// TIA Portal V16 export
// export: Created 2021-12-08T06:27:39.9823919Z, ExportSetting WithDefaults, DisplayName Totally Integrated Automation Portal, DisplayVersion V16 Update 4, DisplayName TIA Portal Version Control Interface, DisplayVersion V16 Update 2, DisplayName TIA Portal Openness, DisplayVersion V16 Update 4, DisplayName TIA Portal Teamcenter Gateway, DisplayVersion V16, DisplayName SINAMICS Startdrive Advanced, DisplayVersion V16 Update 5, DisplayName SINAMICS Startdrive G130, G150, S120, S150, SINAMICS MV, S210, DisplayVersion V16 Update 5, DisplayName SINAMICS Startdrive G110M, G120, G120C, G120D, G120P, G115D, DisplayVersion V16 Update 5, DisplayName STEP 7 Professional, DisplayVersion V16 Update 4, DisplayName STEP 7 Safety, DisplayVersion V16, DisplayName WinCC Advanced, DisplayVersion V16 Update 4
FUNCTION_BLOCK "FB_LexiumModbusTCP"   // FB301, FBD
{ S7_Optimized_Access := 'TRUE' }
VERSION : 0.1
// stored: AutoNumber false, IsIECCheckEnabled false, IsRetainMemResEnabled false, MemoryReserve 100, SetENOAutomatically false, UDAEnableTagReadback false
   VAR_INPUT
      IP_OCTET_01 : USInt;
      IP_OCTET_2 : USInt;
      IP_OCTET_3 : USInt;
      IP_OCTET_4 : USInt;
      ConnectID_1 : CONN_OUC;
      ConnectID_2 : CONN_OUC;
      ConnectID_3 : CONN_OUC;
      ConnectID_4 : CONN_OUC;
      vix_DriveEnable : Bool;
      "vir_Increment/Meter" : Real;
      vix_ExecuteCalib : Bool;
      vii_CalibPos : Int;
      vir_Offset : Real;
      vix_OffsetEnable : Bool;
      vir_RequestPosition_mm : Real;
      vix_ExecuteAutomatic : Bool;
      vii_nVSlow : Int;
      vii_nVFast : Int := 0;
      vii_nVManual : Int := 0;
      vir_nTolerancePosition : Real := 0.0;
      vix_ManualBigger : Bool;
      vix_ManualSmaller : Bool;
      vir_MaxFormat_mm : Real;
      vir_MinFormat_mm : Real;
      vix_ManualParameterDownload : Bool;
      vix_QuickStop : Bool;
      vix_FaultReset : Bool;
   END_VAR
   VAR_OUTPUT
      vix_DriveState : Byte;
      vqx_ComOk : Bool;
      vqx_ReferenceOK : Bool;
      vqx_Error : Bool;
      vqr_ActualPosition_mm : Real;
      vqx_PositionReached : Bool;
      vqx_SoftLimitMAX : Bool;
      vqx_SoftLimitMIN : Bool;
      vqx_SwitchedOn : Bool;
      vqx_DriveFault : Bool;
      vqx_QickStopActive : Bool;
   END_VAR
   VAR_IN_OUT
      ILE_ParameterDB : "ILE1B_Parameter";
      viqr_nToleranceVSlow : Real := 0.0;
      viqr_nToleranceVFast : Real := 0.0;
   END_VAR
   VAR
      Axis_Ref { S7_SetPoint := 'True'} : "ILx2T_Ref";
      ILx2_ModbusTCP_Data_Instance { S7_SetPoint := 'True'} : "ILx2_ModbusTCP_Data";
      ILx2T_Control_Instance { S7_SetPoint := 'True'} : "ILx2T_Control";
      ILx2T_Homing_Instance { S7_SetPoint := 'True'} : "ILx2T_Homing";
      ILx2T_Jog_Instance { S7_SetPoint := 'True'} : "ILx2T_Jog";
      ILx2T_ProfilePosition_Instance { S7_SetPoint := 'True'} : "ILx2T_ProfilePosition";
      ILx2T_ProfileVelocity_Instance { S7_SetPoint := 'True'} : "ILx2T_ProfileVelocity";
      ILx2T_Parameter_Read_Write_Instance { S7_SetPoint := 'True'} : "ILx2T_Parameter_Read_Write";
      ILx2T_SetAcceleration { S7_SetPoint := 'True'} : "ILx2T_Parameter_Read_Write";
      ILx2T_SetDeceleration { S7_SetPoint := 'True'} : "ILx2T_Parameter_Read_Write";
      ILx2T_ReadActualPosition { S7_SetPoint := 'True'} : "ILx2T_Parameter_Read_Write";
      ILx2T_ReadActualVelocity { S7_SetPoint := 'True'} : "ILx2T_Parameter_Read_Write";
      vsx_ComError { S7_SetPoint := 'True'} : Bool;
      vsx_HomeError : Bool;
      vsx_JogError : Bool;
      vsx_PositionError : Bool;
      vsx_VelocityError : Bool;
      vsx_ReadWriteError1 : Bool;
      vsx_ReadWriteError2 : Bool;
      vsx_ReadWriteError3 : Bool;
      vsx_ReadWriteError4 : Bool;
      vsx_ReadWriteError5 : Bool;
      vsr_HomeRefAppPos : Real;
      vqr_RequestPosplusOffset : Real;
      vsr_RequestPosPlusOffsetLimited : Real;
      vqw_StopFaulthex : DWord;
      tmpExecuteAutoSet : Bool;
      tmpRangeMin { ExternalAccessible := 'False'; ExternalVisible := 'False'; ExternalWritable := 'False'} : Real;
      tmpRangeMax { ExternalAccessible := 'False'; ExternalVisible := 'False'; ExternalWritable := 'False'} : Real;
      P_Trig_ComOK : Bool;
      vsx_SetValueOutOfRange : Bool;
      TimerOffsetCorrectino : IEC_TIMER;
      TimerDelayParamterDownload { S7_SetPoint := 'True'} : IEC_TIMER;
      fbMaticExt_Instance { S7_SetPoint := 'True'} : "fbMaticExt";
      TargetVelocity { S7_SetPoint := 'True'} : Int;
      vsi_AcutalPosInc : DInt;
      Testbit : Bool;
   END_VAR
BEGIN

REGION Network 1: Error
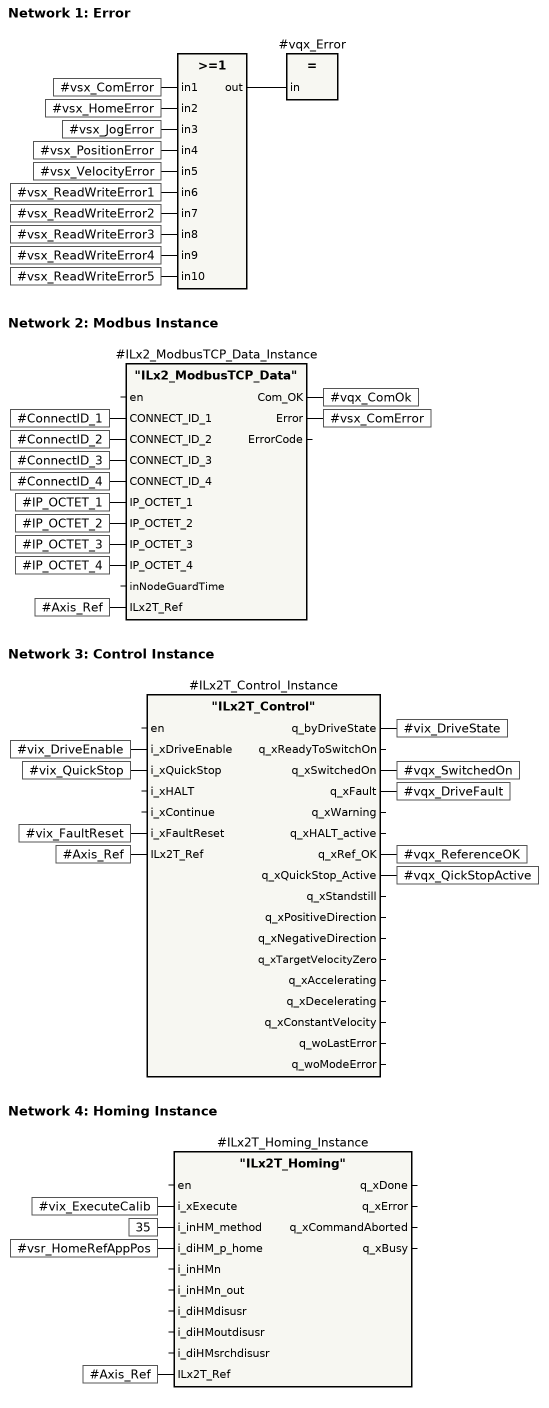
   #vqx_Error := #vsx_ComError OR #vsx_HomeError OR #vsx_JogError OR #vsx_PositionError OR #vsx_VelocityError OR #vsx_ReadWriteError1 OR #vsx_ReadWriteError2 OR #vsx_ReadWriteError3 OR #vsx_ReadWriteError4 OR #vsx_ReadWriteError5;
END_REGION

REGION Network 2: Modbus Instance
   // Error ID -TIA online help (MB_CLIENT)
   #ILx2_ModbusTCP_Data_Instance(CONNECT_ID_1 := #ConnectID_1,   // "ILx2_ModbusTCP_Data"
                           CONNECT_ID_2 := #ConnectID_2,
                           CONNECT_ID_3 := #ConnectID_3,
                           CONNECT_ID_4 := #ConnectID_4,
                           IP_OCTET_1 := #IP_OCTET_1,
                           IP_OCTET_2 := #IP_OCTET_2,
                           IP_OCTET_3 := #IP_OCTET_3,
                           IP_OCTET_4 := #IP_OCTET_4,
                           ILx2T_Ref := #Axis_Ref,
                           Com_OK => #vqx_ComOk,
                           Error => #vsx_ComError);
END_REGION

REGION Network 3: Control Instance
   #ILx2T_Control_Instance(i_xDriveEnable := #vix_DriveEnable,   // "ILx2T_Control"
                           i_xQuickStop := #vix_QuickStop,
                           i_xFaultReset := #vix_FaultReset,
                           ILx2T_Ref := #Axis_Ref,
                           q_byDriveState => #vix_DriveState,
                           q_xSwitchedOn => #vqx_SwitchedOn,
                           q_xFault => #vqx_DriveFault,
                           q_xRef_OK => #vqx_ReferenceOK,
                           q_xQuickStop_Active => #vqx_QickStopActive);
END_REGION

REGION Network 4: Homing Instance
   #ILx2T_Homing_Instance(i_xExecute := #vix_ExecuteCalib,   // "ILx2T_Homing"
                          i_inHM_method := 35,
                          i_diHM_p_home := #vsr_HomeRefAppPos,
                          ILx2T_Ref := #Axis_Ref);
END_REGION

REGION Network 5: Jog Instance (Not Used)
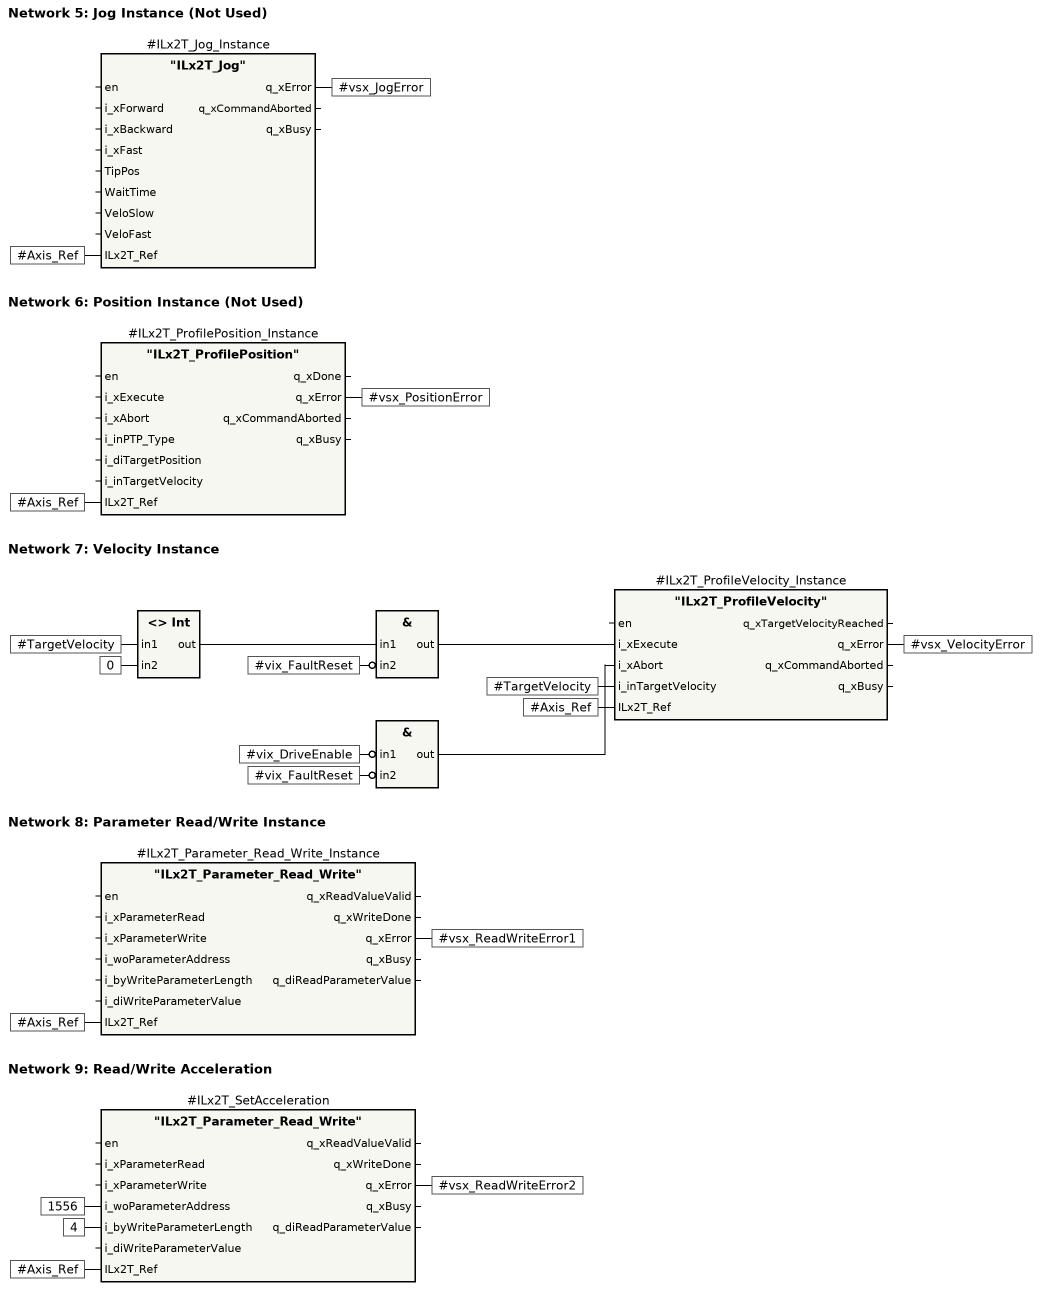
   #ILx2T_Jog_Instance(ILx2T_Ref := #Axis_Ref, q_xError => #vsx_JogError);   // "ILx2T_Jog"
END_REGION

REGION Network 6: Position Instance (Not Used)
   #ILx2T_ProfilePosition_Instance(ILx2T_Ref := #Axis_Ref, q_xError => #vsx_PositionError);   // "ILx2T_ProfilePosition"
END_REGION

REGION Network 7: Velocity Instance
   #ILx2T_ProfileVelocity_Instance(i_xExecute := (#TargetVelocity <> 0) AND NOT #vix_FaultReset,   // "ILx2T_ProfileVelocity"
                           i_xAbort := NOT #vix_DriveEnable AND NOT #vix_FaultReset,
                           i_inTargetVelocity := #TargetVelocity,
                           ILx2T_Ref := #Axis_Ref,
                           q_xError => #vsx_VelocityError);
END_REGION

REGION Network 8: Parameter Read/Write Instance
   #ILx2T_Parameter_Read_Write_Instance(ILx2T_Ref := #Axis_Ref, q_xError => #vsx_ReadWriteError1);   // "ILx2T_Parameter_Read_Write"
END_REGION

REGION Network 9: Read/Write Acceleration
   #ILx2T_SetAcceleration(i_woParameterAddress := 1556,   // "ILx2T_Parameter_Read_Write"
                          i_byWriteParameterLength := 4,
                          ILx2T_Ref := #Axis_Ref,
                          q_xError => #vsx_ReadWriteError2);
END_REGION

REGION Network 10: Read/Write Deceleration
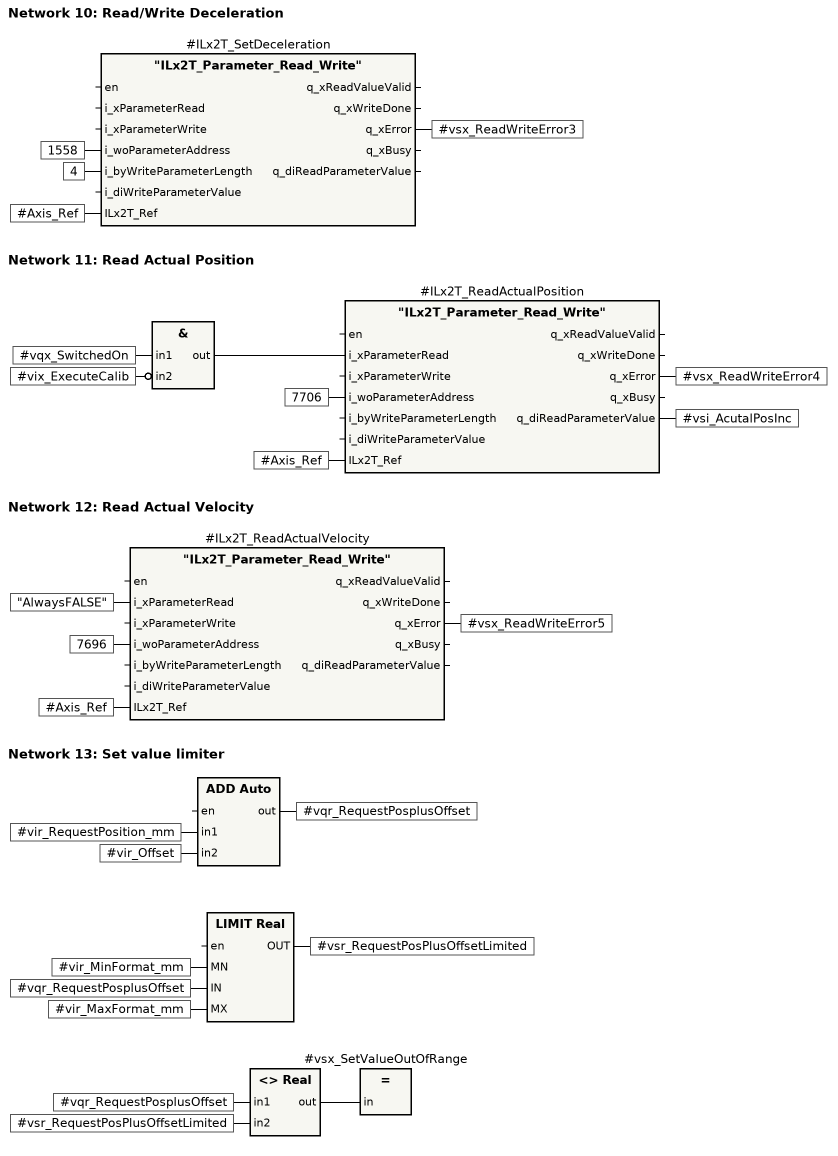
   #ILx2T_SetDeceleration(i_woParameterAddress := 1558,   // "ILx2T_Parameter_Read_Write"
                          i_byWriteParameterLength := 4,
                          ILx2T_Ref := #Axis_Ref,
                          q_xError => #vsx_ReadWriteError3);
END_REGION

REGION Network 11: Read Actual Position
   #ILx2T_ReadActualPosition(i_xParameterRead := #vqx_SwitchedOn AND NOT #vix_ExecuteCalib,   // "ILx2T_Parameter_Read_Write"
                           i_woParameterAddress := 7706,
                           ILx2T_Ref := #Axis_Ref,
                           q_xError => #vsx_ReadWriteError4,
                           q_diReadParameterValue => #vsi_AcutalPosInc);
END_REGION

REGION Network 12: Read Actual Velocity
   #ILx2T_ReadActualVelocity(i_xParameterRead := "AlwaysFALSE",   // "ILx2T_Parameter_Read_Write"
                           i_woParameterAddress := 7696,
                           ILx2T_Ref := #Axis_Ref,
                           q_xError => #vsx_ReadWriteError5);
END_REGION

REGION Network 13: Set value limiter
   #vqr_RequestPosplusOffset := #vir_RequestPosition_mm + #vir_Offset;
   #vsr_RequestPosPlusOffsetLimited := LIMIT(MN := #vir_MinFormat_mm, IN := #vqr_RequestPosplusOffset, MX := #vir_MaxFormat_mm);
   #vsx_SetValueOutOfRange := #vqr_RequestPosplusOffset <> #vsr_RequestPosPlusOffsetLimited;
END_REGION

REGION Network 14: Matic Module
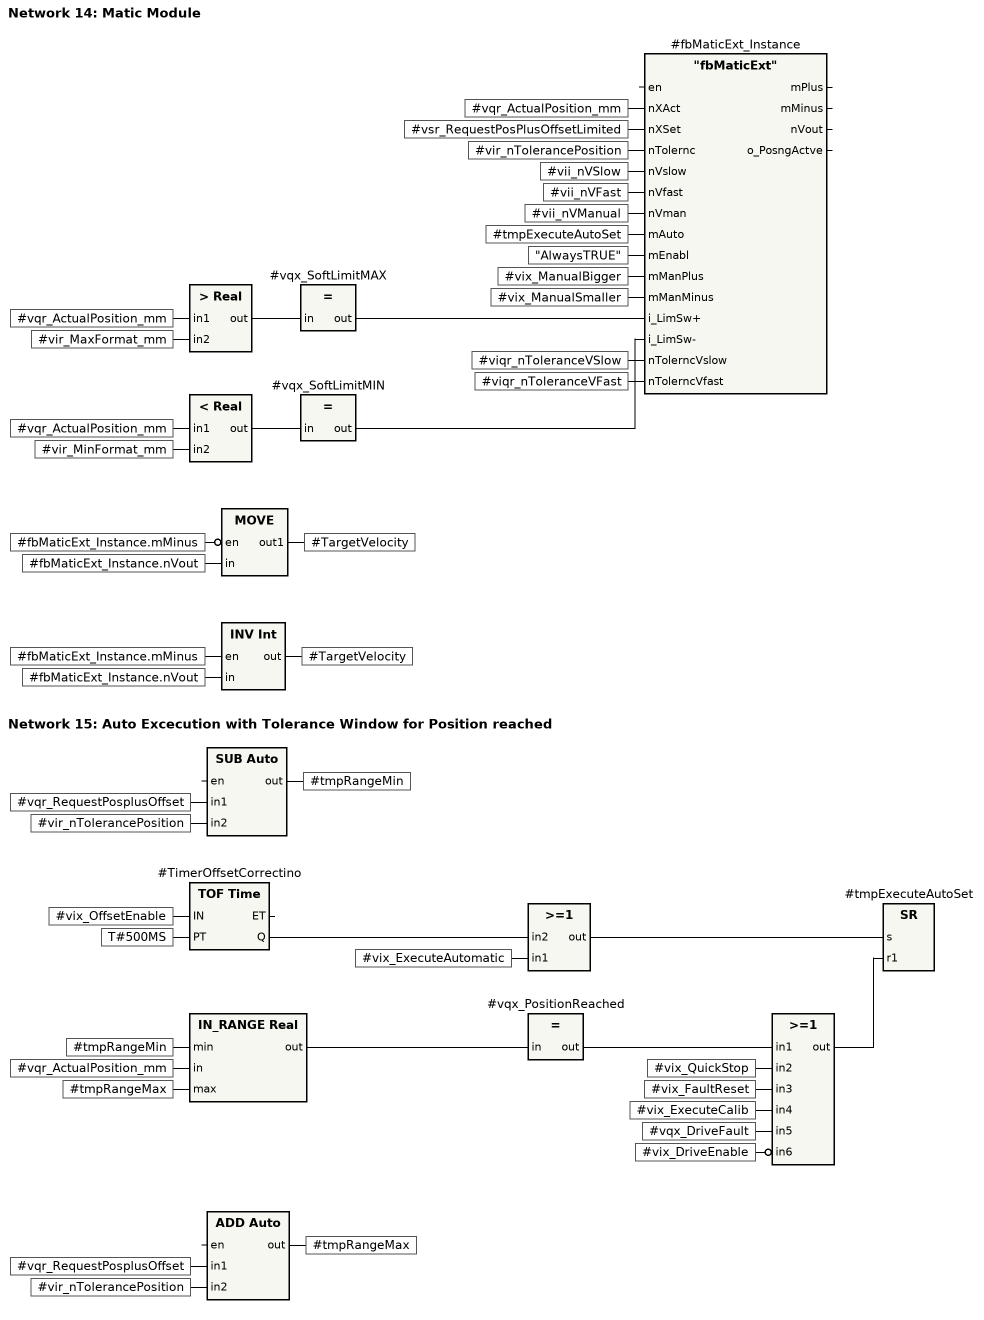
   #vqx_SoftLimitMAX := #vqr_ActualPosition_mm > #vir_MaxFormat_mm;
   #vqx_SoftLimitMIN := #vqr_ActualPosition_mm < #vir_MinFormat_mm;
   #fbMaticExt_Instance(nXAct := #vqr_ActualPosition_mm,   // "fbMaticExt"
                        nXSet := #vsr_RequestPosPlusOffsetLimited,
                        nTolernc := #vir_nTolerancePosition,
                        nVslow := #vii_nVSlow,
                        nVfast := #vii_nVFast,
                        nVman := #vii_nVManual,
                        mAuto := #tmpExecuteAutoSet,
                        mEnabl := "AlwaysTRUE",
                        mManPlus := #vix_ManualBigger,
                        mManMinus := #vix_ManualSmaller,
                        "i_LimSw+" := #vqx_SoftLimitMAX,
                        "i_LimSw-" := #vqx_SoftLimitMIN,
                        nTolerncVslow := #viqr_nToleranceVSlow,
                        nTolerncVfast := #viqr_nToleranceVFast);
   IF NOT #fbMaticExt_Instance.mMinus THEN #TargetVelocity := #fbMaticExt_Instance.nVout; END_IF;
   IF #fbMaticExt_Instance.mMinus THEN #TargetVelocity := NOT #fbMaticExt_Instance.nVout; END_IF;
END_REGION

REGION Network 15: Auto Excecution with Tolerance Window for Position reached
   #tmpRangeMin := #vqr_RequestPosplusOffset - #vir_nTolerancePosition;
   #TimerOffsetCorrectino.TOF(IN := #vix_OffsetEnable, PT := T#500MS);
   #vqx_PositionReached := (#tmpRangeMin <= #vqr_ActualPosition_mm) AND (#vqr_ActualPosition_mm <= #tmpRangeMax);
   IF #TimerOffsetCorrectino.Q OR #vix_ExecuteAutomatic THEN
       #tmpExecuteAutoSet := TRUE;   // SR flip-flop
   END_IF;
   IF #vqx_PositionReached OR #vix_QuickStop OR #vix_FaultReset OR #vix_ExecuteCalib OR #vqx_DriveFault OR NOT #vix_DriveEnable THEN
       #tmpExecuteAutoSet := FALSE;
   END_IF;
   #tmpRangeMax := #vqr_RequestPosplusOffset + #vir_nTolerancePosition;
END_REGION

REGION Network 16: Scaling Increment in mm
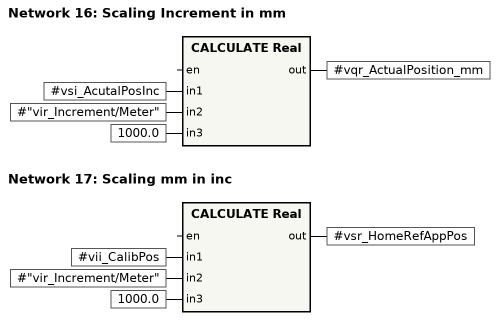
   #vqr_ActualPosition_mm := #vsi_AcutalPosInc * (#"vir_Increment/Meter"/1000.0);
END_REGION

REGION Network 17: Scaling mm in inc
   #vsr_HomeRefAppPos := #vii_CalibPos/(#"vir_Increment/Meter"/1000.0);
END_REGION
END_FUNCTION_BLOCK
